Yaskawa INFORM job: TEST_LASER.JBI

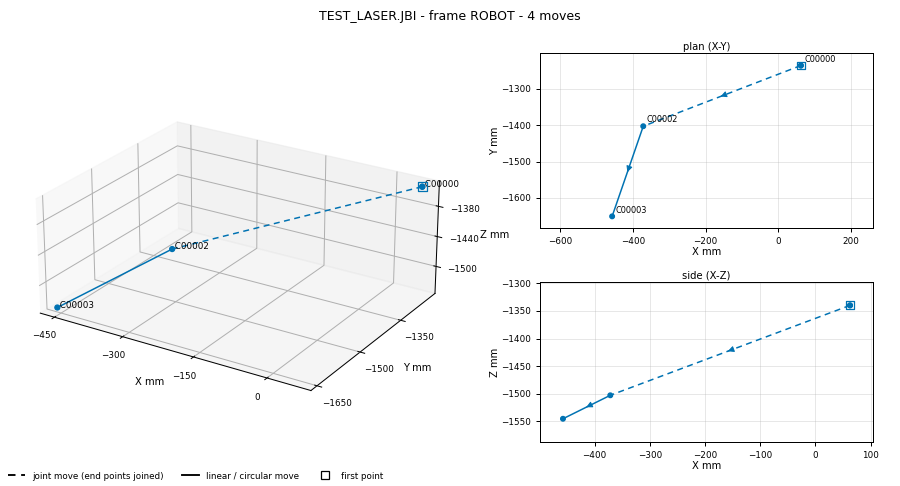
[picture p0: tool path of TEST_LASER.JBI in frame ROBOT, 4 of 4 moves have a stored position in this frame; points joined in program order, loops and branches not executed]
/JOB
//NAME TEST_LASER
//POS
///NPOS 4,4,0,0,0,0
///TOOL 0
///POSTYPE ROBOT
///RECTAN
///RCONF 0,0,0,0,1,0,0,0,0,0,0,0,0,0,0,0,0,0,0,0,0,0,0,0
C00000=62.554,-1235.469,-1339.933,-0.1773,5.3581,-86.9836
///RCONF 0,0,0,0,0,0,0,0,0,0,0,0,0,0,0,0,0,0,0,0,0,0,0,0
C00001=62.548,-1235.474,-1339.938,-49.3265,-2.1593,-90.0984
C00002=-371.677,-1402.690,-1502.805,-49.3259,-2.1593,-90.0974
C00003=-457.402,-1650.966,-1545.305,-47.1489,-2.1778,-89.5609
BC00000=2441.469,2554.202,758.861
BC00001=2441.469,2554.202,758.861
BC00002=2441.469,2554.202,758.861
BC00003=2441.469,2554.202,758.861
//INST
///DATE 2023/11/02 14:32
///ATTR SC,RW,RJ
////FRAME ROBOT
///GROUP1 RB1,BS1
NOP
MOVJ C00000 BC00000 VJ=20.00
MOVJ C00001 BC00001 VJ=20.00
MOVJ C00002 BC00002 VJ=20.00
ARCON
MOVL C00003 BC00003 V=11.0
END
